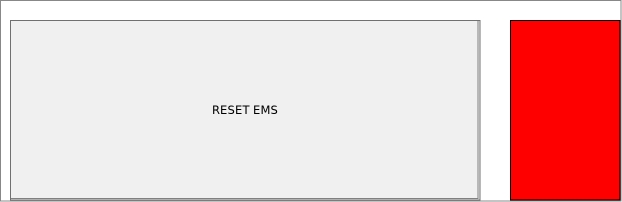
VISUALIZATION Visu1  // 622x202
    Button (10,20 470x180), "RESET EMS"
        tap Global_IOs.PC_RESET_EMS
    Rectangle (510,20 110x180), colour toggle: Global_IOs.EMS_OK
END_VISUALIZATION

(* stored: Version 1.1.0.1, ProductVersion 3.1.0.26
   Visu Visu1: Id {d51c156c-3f8e-4364-9dbb-0f429427b319} *)
